// TIA Portal V19 export
TYPE "MachineInterface"
// stored: Access Published
   STRUCT
      AutReady : Bool;   // Lower Dead Point / Machine ready for automatic cycle
      Aborting : Bool;   // Machine must stay in Normal Stop During Restart / Machine is aborting (alarm presence)
      AckStopInPhase : Bool;   // Stop cycle for aborting / Machine ack to area stop in phase
      AckStopProgrammed : Bool;   // Stop cycle programmed has been done / Machine ack to area stop programmed
      MotionsStandStill : Bool;   // Alarms Synch sensor (table) not catch / loose / Machine motion Standstill
      AlarmsPresence : Bool;   // Alarms & Mesage Out / Machine alarms presence (for lamp signaling)
      WarningPresence : Bool;   // Warnings / Machine warnings presence (for lamp signaling)
   END_STRUCT;
END_TYPE
